Universal Robots PolyScope program: movej_l_p_v2.urp

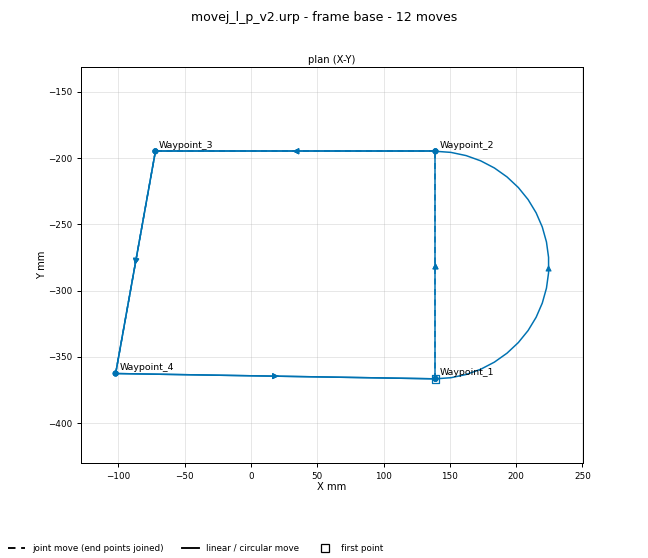
[picture p0: tool path of movej_l_p_v2.urp in frame base, 12 of 13 moves have a stored position in this frame; points joined in program order, loops and branches not executed]
Program movej_l_p_v2 (installation=default directory=/home/ur/ursim-current/programs createdIn=3.6.1.30595 lastSavedIn=3.14.3.1031232 robotSerialNumber=2018339999)
Calibrated DH parameters: a=[0, -0.24365, -0.21325, 0, 0, 0]; d=[0.1519, 0, 0, 0.11235, 0.08535, 0.0819]; alpha=[1.570796, 0, 0, 1.570796, -1.570796, 0]; deltaTheta=[0, 0, 0, 0, 0, 0]
Robot Program (runOnlyOnce=false)
  MoveJ speed 60 deg/s, acceleration 80 deg/s^2 (useActiveTCP=true)
    Waypoint Waypoint_1: TCP in base x=139.155 y=-366.472 z=77.328 mm, rx=-0.0012 ry=3.1163 rz=0.0389 rad; joints [-53.415, -119.404, -96.349, -54.54, 92.006, 36.535] deg; flange x=137.15 y=-368.469 z=157.278 mm, rx=-0.0012 ry=3.1163 rz=0.0389 rad
    Waypoint Waypoint_2: TCP in base x=139.155 y=-194.881 z=77.328 mm, rx=-0.0012 ry=3.1163 rz=0.0389 rad; joints [-27.235, -116.144, -148.658, -4.576, 91.929, 62.731] deg
    Waypoint Waypoint_3: TCP in base x=-72.037 y=-194.881 z=77.328 mm, rx=-0.0012 ry=3.1163 rz=0.0389 rad; joints [-79.096, -76.17, -147.657, -47.307, 91.681, 10.843] deg; flange x=-74.042 y=-196.878 z=157.278 mm, rx=-0.0012 ry=3.1163 rz=0.0389 rad
    Waypoint Waypoint_4: TCP in base x=-102.037 y=-362.472 z=77.328 mm, rx=-0.0012 ry=3.1163 rz=0.0389 rad; joints [-89.02, -116.613, -100.447, -54.346, 91.46, 0.918] deg; flange x=-104.042 y=-364.469 z=157.278 mm, rx=-0.0012 ry=3.1163 rz=0.0389 rad
  MoveL speed 250 mm/s, acceleration 1200 mm/s^2 (useActiveTCP=true) feature=Base
    Waypoint Waypoint_1: TCP in base x=139.155 y=-366.472 z=77.328 mm, rx=-0.0012 ry=3.1163 rz=0.0389 rad; joints [-53.415, -119.404, -96.349, -54.54, 92.006, 36.535] deg; flange x=137.15 y=-368.469 z=157.278 mm, rx=-0.0012 ry=3.1163 rz=0.0389 rad
    Waypoint Waypoint_2: TCP in base x=139.155 y=-194.881 z=77.328 mm, rx=-0.0012 ry=3.1163 rz=0.0389 rad; joints [-27.235, -116.144, -148.658, -4.576, 91.929, 62.731] deg
    Waypoint Waypoint_3: TCP in base x=-72.037 y=-194.881 z=77.328 mm, rx=-0.0012 ry=3.1163 rz=0.0389 rad; joints [-79.096, -76.17, -147.657, -47.307, 91.681, 10.843] deg; flange x=-74.042 y=-196.878 z=157.278 mm, rx=-0.0012 ry=3.1163 rz=0.0389 rad
    Waypoint Waypoint_4: TCP in base x=-102.037 y=-362.472 z=77.328 mm, rx=-0.0012 ry=3.1163 rz=0.0389 rad; joints [-89.02, -116.613, -100.447, -54.346, 91.46, 0.918] deg; flange x=-104.042 y=-364.469 z=157.278 mm, rx=-0.0012 ry=3.1163 rz=0.0389 rad
  MoveP speed 250 mm/s, acceleration 1200 mm/s^2 (blendRadius=0.025 useActiveTCP=true) feature=Base
    Waypoint Waypoint_1: TCP in base x=139.155 y=-366.472 z=77.328 mm, rx=-0.0012 ry=3.1163 rz=0.0389 rad; joints [-53.415, -119.404, -96.349, -54.54, 92.006, 36.535] deg; flange x=137.15 y=-368.469 z=157.278 mm, rx=-0.0012 ry=3.1163 rz=0.0389 rad
    CircleMove (OrientationMode=FIXED)
      Waypoint ViaPoint_1: TCP in base x=224.497 y=-285.457 z=77.328 mm, rx=-0.0012 ry=3.1163 rz=0.0389 rad; joints [-34.728, -113.494, -106.399, -49.741, 91.994, 55.234] deg; flange x=222.493 y=-287.454 z=157.278 mm, rx=-0.0012 ry=3.1163 rz=0.0389 rad
      Waypoint EndPoint_1: TCP in base x=139.155 y=-194.881 z=77.328 mm, rx=-0.0012 ry=3.1163 rz=0.0389 rad; joints [-27.963, -85.906, -141.382, -42.113, 91.937, 62.002] deg; flange x=137.15 y=-196.878 z=157.278 mm, rx=-0.0012 ry=3.1163 rz=0.0389 rad
    SuppressedNode
      Waypoint Waypoint_2: motionParameters(jointSpeed=1.047198 jointAcceleration=1.396263 cartesianSpeed=0.25 cartesianAcceleration=1.2 blendRadius=0); TCP in base x=139.155 y=-194.881 z=77.328 mm, rx=-0.0012 ry=3.1163 rz=0.0389 rad; joints [-27.235, -116.144, -148.658, -4.576, 91.929, 62.731] deg
    Waypoint Waypoint_3: TCP in base x=-72.037 y=-194.881 z=77.328 mm, rx=-0.0012 ry=3.1163 rz=0.0389 rad; joints [-79.096, -76.17, -147.657, -47.307, 91.681, 10.843] deg; flange x=-74.042 y=-196.878 z=157.278 mm, rx=-0.0012 ry=3.1163 rz=0.0389 rad
    Waypoint Waypoint_4: TCP in base x=-102.037 y=-362.472 z=77.328 mm, rx=-0.0012 ry=3.1163 rz=0.0389 rad; joints [-89.02, -116.613, -100.447, -54.346, 91.46, 0.918] deg; flange x=-104.042 y=-364.469 z=157.278 mm, rx=-0.0012 ry=3.1163 rz=0.0389 rad
